% RSLogix 500 project Project 10.RSS, saved by version 8.30.00.16 %
PROJECT "UNTITLED"    % processor: Bul.1763 MicroLogix 1100 Series B %

PROGRAM FILES
  LAD 2 "MAIN"  5 rungs
  LAD 3 "IO"  8 rungs
  LAD 4 "CONTROLS"  7 rungs
  LAD 5 "ALARMS"  9 rungs
  LAD 6 "HOA"  6 rungs

DATA FILES
  O0 OUTPUT  4 elements
  I1 INPUT  6 elements
  S2 STATUS  66 elements
  B3 BINARY  2 elements
  T4 TIMER  4 elements
  C5 COUNTER  1 elements
  R6 CONTROL  1 elements
  N7 INTEGER  4 elements
  F8 FLOAT  1 elements

LADDER 2 "MAIN"
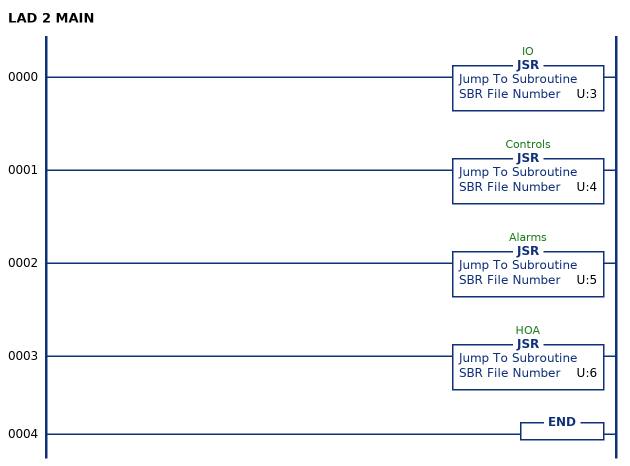
% Rung: 0 %
SOR JSR U:3 EOR
%   U:3  "IO" %
% Rung: 1 %
SOR JSR U:4 EOR
%   U:4  "Controls" %
% Rung: 2 %
SOR JSR U:5 EOR
%   U:5  "Alarms" %
% Rung: 3 %
SOR JSR U:6 EOR
%   U:6  "HOA" %
% Rung: 4 %
SOR END EOR

LADDER 3 "IO"
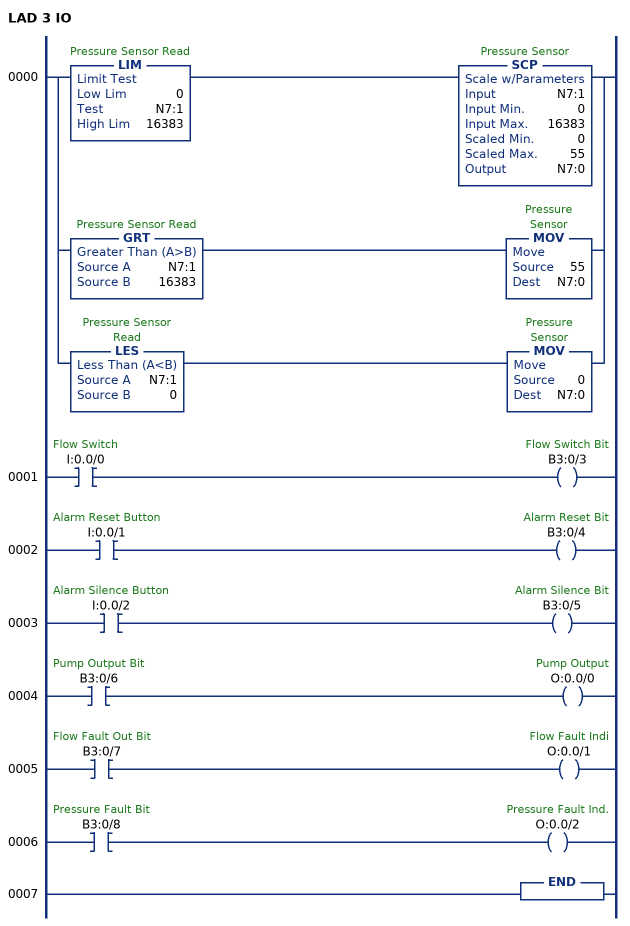
% Rung: 0 %
SOR BST LIM 0 N7:1 16383 SCP N7:1 0 16383 0 55 N7:0 NXB GRT N7:1 16383 MOV 55 N7:0 NXB LES N7:1 0 MOV 0 N7:0 BND EOR
%   N7:1  "Pressure Sensor Read" %
%   N7:0  "Pressure Sensor" %
% Rung: 1 %
SOR XIC I:0.0/0 OTE B3:0/3 EOR
%   I:0.0/0  "Flow Switch" %
%   B3:0/3  "Flow Switch Bit" %
% Rung: 2 %
SOR XIC I:0.0/1 OTE B3:0/4 EOR
%   I:0.0/1  "Alarm Reset Button" %
%   B3:0/4  "Alarm Reset Bit" %
% Rung: 3 %
SOR XIC I:0.0/2 OTE B3:0/5 EOR
%   I:0.0/2  "Alarm Silence Button" %
%   B3:0/5  "Alarm Silence Bit" %
% Rung: 4 %
SOR XIC B3:0/6 OTE O:0.0/0 EOR
%   B3:0/6  "Pump Output Bit" %
%   O:0.0/0  "Pump Output" %
% Rung: 5 %
SOR XIC B3:0/7 OTE O:0.0/1 EOR
%   B3:0/7  "Flow Fault Out Bit" %
%   O:0.0/1  "Flow Fault Indi" %
% Rung: 6 %
SOR XIC B3:0/8 OTE O:0.0/2 EOR
%   B3:0/8  "Pressure Fault Bit" %
%   O:0.0/2  "Pressure Fault Ind." %
% Rung: 7 %
SOR END EOR

LADDER 4 "CONTROLS"
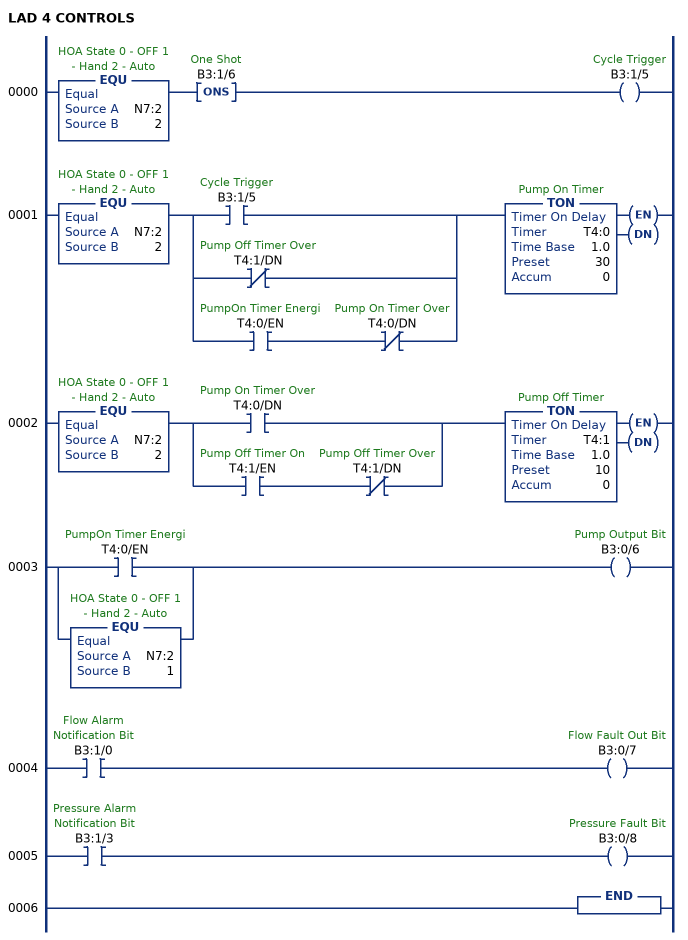
% Rung: 0 %
SOR EQU N7:2 2 ONS B3:1/6 OTE B3:1/5 EOR
%   N7:2  "HOA State 0 - OFF 1 - Hand 2 - Auto" %
%   B3:1/6  "One Shot" %
%   B3:1/5  "Cycle Trigger" %
% Rung: 1 %
SOR EQU N7:2 2 BST XIC B3:1/5 NXB XIO T4:1/DN NXB XIC T4:0/EN XIO T4:0/DN BND TON T4:0 1.0 30 0 EOR
%   N7:2  "HOA State 0 - OFF 1 - Hand 2 - Auto" %
%   B3:1/5  "Cycle Trigger" %
%   T4:1/DN  "Pump Off Timer Over" %
%   T4:0/EN  "PumpOn Timer Energi" %
%   T4:0/DN  "Pump On Timer Over" %
%   T4:0  "Pump On Timer" %
% Rung: 2 %
SOR EQU N7:2 2 BST XIC T4:0/DN NXB XIC T4:1/EN XIO T4:1/DN BND TON T4:1 1.0 10 0 EOR
%   N7:2  "HOA State 0 - OFF 1 - Hand 2 - Auto" %
%   T4:0/DN  "Pump On Timer Over" %
%   T4:1/EN  "Pump Off Timer On" %
%   T4:1/DN  "Pump Off Timer Over" %
%   T4:1  "Pump Off Timer" %
% Rung: 3 %
SOR BST XIC T4:0/EN NXB EQU N7:2 1 BND OTE B3:0/6 EOR
%   T4:0/EN  "PumpOn Timer Energi" %
%   N7:2  "HOA State 0 - OFF 1 - Hand 2 - Auto" %
%   B3:0/6  "Pump Output Bit" %
% Rung: 4 %
SOR XIC B3:1/0 OTE B3:0/7 EOR
%   B3:1/0  "Flow Alarm Notification Bit" %
%   B3:0/7  "Flow Fault Out Bit" %
% Rung: 5 %
SOR XIC B3:1/3 OTE B3:0/8 EOR
%   B3:1/3  "Pressure Alarm Notification Bit" %
%   B3:0/8  "Pressure Fault Bit" %
% Rung: 6 %
SOR END EOR

LADDER 5 "ALARMS"
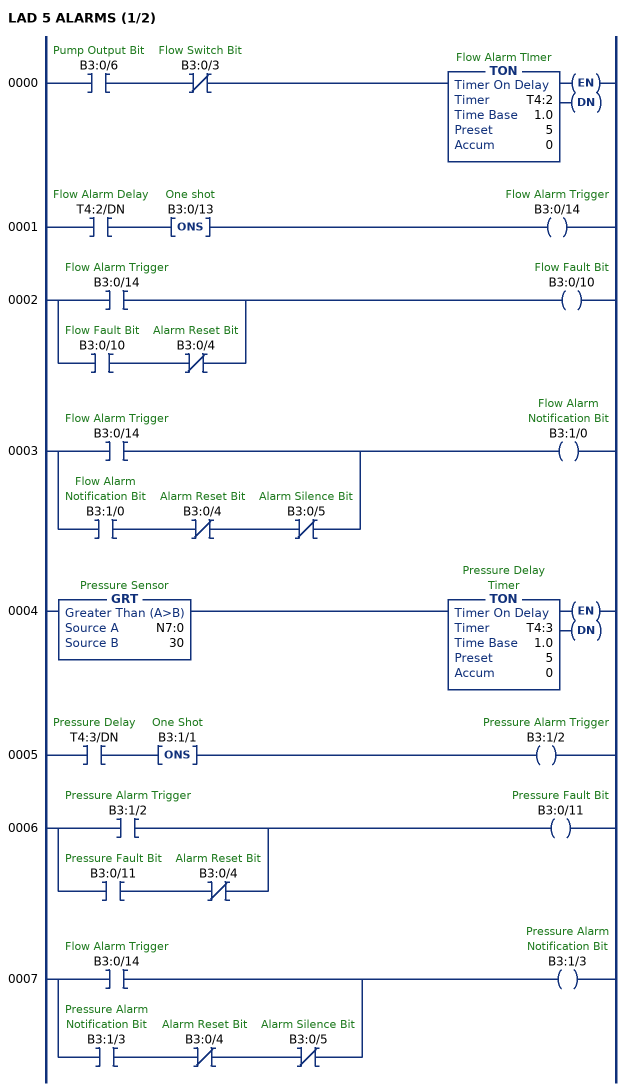
% Rung: 0 %
SOR XIC B3:0/6 XIO B3:0/3 TON T4:2 1.0 5 0 EOR
%   B3:0/6  "Pump Output Bit" %
%   B3:0/3  "Flow Switch Bit" %
%   T4:2  "Flow Alarm TImer" %
% Rung: 1 %
SOR XIC T4:2/DN ONS B3:0/13 OTE B3:0/14 EOR
%   T4:2/DN  "Flow Alarm Delay" %
%   B3:0/13  "One shot" %
%   B3:0/14  "Flow Alarm Trigger" %
% Rung: 2 %
SOR BST XIC B3:0/14 NXB XIC B3:0/10 XIO B3:0/4 BND OTE B3:0/10 EOR
%   B3:0/14  "Flow Alarm Trigger" %
%   B3:0/10  "Flow Fault Bit" %
%   B3:0/4  "Alarm Reset Bit" %
% Rung: 3 %
SOR BST XIC B3:0/14 NXB XIC B3:1/0 XIO B3:0/4 XIO B3:0/5 BND OTE B3:1/0 EOR
%   B3:0/14  "Flow Alarm Trigger" %
%   B3:1/0  "Flow Alarm Notification Bit" %
%   B3:0/4  "Alarm Reset Bit" %
%   B3:0/5  "Alarm Silence Bit" %
% Rung: 4 %
SOR GRT N7:0 30 TON T4:3 1.0 5 0 EOR
%   N7:0  "Pressure Sensor" %
%   T4:3  "Pressure Delay Timer" %
% Rung: 5 %
SOR XIC T4:3/DN ONS B3:1/1 OTE B3:1/2 EOR
%   T4:3/DN  "Pressure Delay" %
%   B3:1/1  "One Shot" %
%   B3:1/2  "Pressure Alarm Trigger" %
% Rung: 6 %
SOR BST XIC B3:1/2 NXB XIC B3:0/11 XIO B3:0/4 BND OTE B3:0/11 EOR
%   B3:1/2  "Pressure Alarm Trigger" %
%   B3:0/11  "Pressure Fault Bit" %
%   B3:0/4  "Alarm Reset Bit" %
% Rung: 7 %
SOR BST XIC B3:0/14 NXB XIC B3:1/3 XIO B3:0/4 XIO B3:0/5 BND OTE B3:1/3 EOR
%   B3:0/14  "Flow Alarm Trigger" %
%   B3:1/3  "Pressure Alarm Notification Bit" %
%   B3:0/4  "Alarm Reset Bit" %
%   B3:0/5  "Alarm Silence Bit" %

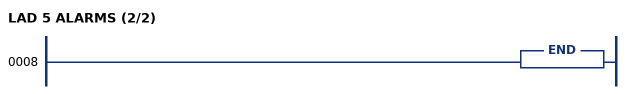
% Rung: 8 %
SOR END EOR

LADDER 6 "HOA"
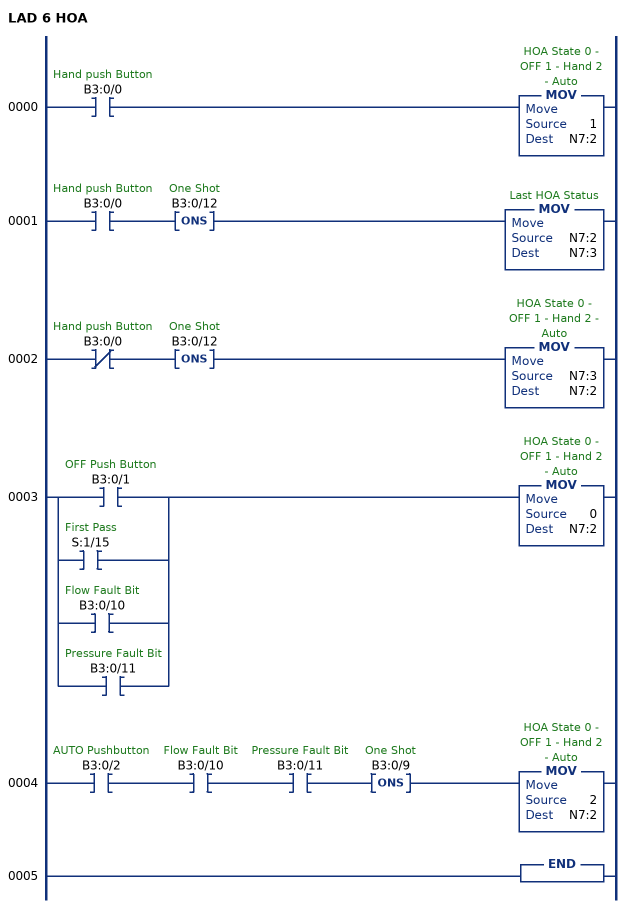
% Rung: 0 %
SOR XIC B3:0/0 MOV 1 N7:2 EOR
%   B3:0/0  "Hand push Button" %
%   N7:2  "HOA State 0 - OFF 1 - Hand 2 - Auto" %
% Rung: 1 %
SOR XIC B3:0/0 ONS B3:0/12 MOV N7:2 N7:3 EOR
%   B3:0/0  "Hand push Button" %
%   B3:0/12  "One Shot" %
%   N7:2  "HOA State 0 - OFF 1 - Hand 2 - Auto" %
%   N7:3  "Last HOA Status" %
% Rung: 2 %
SOR XIO B3:0/0 ONS B3:0/12 MOV N7:3 N7:2 EOR
%   B3:0/0  "Hand push Button" %
%   B3:0/12  "One Shot" %
%   N7:3  "Last HOA Status" %
%   N7:2  "HOA State 0 - OFF 1 - Hand 2 - Auto" %
% Rung: 3 %
SOR BST XIC B3:0/1 NXB XIC S:1/15 NXB XIC B3:0/10 NXB XIC B3:0/11 BND MOV 0 N7:2 EOR
%   B3:0/1  "OFF Push Button" %
%   S:1/15  "First Pass" %
%   B3:0/10  "Flow Fault Bit" %
%   B3:0/11  "Pressure Fault Bit" %
%   N7:2  "HOA State 0 - OFF 1 - Hand 2 - Auto" %
% Rung: 4 %
SOR XIC B3:0/2 XIC B3:0/10 XIC B3:0/11 ONS B3:0/9 MOV 2 N7:2 EOR
%   B3:0/2  "AUTO Pushbutton" %
%   B3:0/10  "Flow Fault Bit" %
%   B3:0/11  "Pressure Fault Bit" %
%   B3:0/9  "One Shot" %
%   N7:2  "HOA State 0 - OFF 1 - Hand 2 - Auto" %
% Rung: 5 %
SOR END EOR

OTHER DOCUMENTED ADDRESSES
  LIM  "Value Check"

DATA TABLE (non-zero values as saved)
DATA T4
% .PRE .ACC %
% T4:0 % 30 0
% T4:1 % 10 0
% T4:2 % 5 0
% T4:3 % 5 0
